PROGRAM MAIN
VAR
END_VAR

END_PROGRAM

(* stored: Version 1.1.0.1
   POU MAIN: Id {52db3fdf-1dfc-4f68-a5da-8fa3c18bf101} *)
